// TIA Portal V20 export
DATA_BLOCK "Instance_FB_Digital_Output_DB"   // DB103
// stored: AutoNumber false, InstanceOfName FB_Digital_Output, InstanceOfType FB
"FB_Digital_Output"
   // VAR_INPUT
   //    DB_In_Emergency_Stop_Release : Bool;
   //    DB_In_Selected_Voltage_220V : Bool;
   //    DB_In_Selected_Voltage_127V : Bool;
   //    DB_Spin_Carousel_Frequency_Inverter_Speed_1 : Bool;
   //    DB_Spin_Carousel_Frequency_Inverter_Speed_2 : Bool;
   //    DB_Spin_Carousel_Frequency_Inverter_Speed_3 : Bool;
   //    DB_Conveyor_Belt_Frequency_Inverter_Speed_1 : Bool;
   //    DB_Conveyor_Belt_Frequency_Inverter_Speed_2 : Bool;
   //    DB_Conveyor_Belt_Frequency_Inverter_Speed_3 : Bool;
   //    DB_Turn_On_Conveyor_Belt_Motor_Spinner_Get_Entrace_Function_Test : Bool;
   //    DB_Turn_On_Conveyor_Belt_Motor_Rework_Conveyor_Belt_Get_Entrace_Functional_Test : Bool;
   //    DB_Turn_On_Conveyor_Belt_Motor_Spinner_Get_Exit_Functional_Test : Bool;
   //    DB_Turn_On_Conveyor_Belt_Motor_Rework_Conveyor_Belt_Get_Exit_Funcional_Test : Bool;
   //    DB_Open_Air_Pressure : Bool;
   //    DB_Valve_Advance_Spinner_Get_Entrace_Functional_Test : Bool;
   //    DB_Valve_Advance_Spinner_Get_Exit_Functional_Test : Bool;
   //    DB_Signal_Pre_Functional_Test_Production_Line : Bool;
   //    DB_Digital_Output_14 : Bool;
   //    DB_Digital_Output_15 : Bool;
   //    DB_Digital_Output_16 : Bool;
   //    DB_Digital_Output_17 : Bool;
   //    DB_Digital_Output_18 : Bool;
   //    DB_Digital_Output_19 : Bool;
   //    DB_Digital_Output_20 : Bool;
   //    DB_Digital_Output_21 : Bool;
   //    DB_Digital_Output_22 : Bool;
   //    DB_Digital_Output_23 : Bool;
   //    DB_Voltage_220V_Selected : Bool;
   //    DB_Voltage_127V_Selected : Bool;
   // END_VAR
   // VAR_OUTPUT
   //    DO_Spin_Carousel_Frequency_Inverter_Speed_1 : Bool;
   //    DO_Spin_Carousel_Frequency_Inverter_Speed_2 : Bool;
   //    DO_Spin_Carousel_Frequency_Inverter_Speed_3 : Bool;
   //    DO_Conveyor_Belt_Frequency_Inverter_Speed_1 : Bool;
   //    DO_Conveyor_Belt_Frequency_Inverter_Speed_2 : Bool;
   //    DO_Conveyor_Belt_Frequency_Inverter_Speed_3 : Bool;
   //    DO_Turn_On_Conveyor_Belt_Motor_Spinner_Get_Entrace_Function_Test : Bool;
   //    DO_Turn_On_Conveyor_Belt_Motor_Rework_Conveyor_Belt_Get_Entrace_Functional_Test : Bool;
   //    DO_Turn_On_Conveyor_Belt_Motor_Spinner_Get_Exit_Functional_Test : Bool;
   //    DO_Turn_On_Conveyor_Belt_Motor_Rework_Conveyor_Belt_Get_Exit_Funcional_Test : Bool;
   //    DO_Open_Air_Pressure : Bool;
   //    DO_Valve_Advance_Spinner_Entrace_Functional_Test : Bool;
   //    DO_Valve_Advance_Spinner_Exit_Functional_Test : Bool;
   //    DO_Signal_Pre_Functional_Test_Production_Line : Bool;
   //    DO_Digital_Output_14 : Bool;
   //    DO_Digital_Output_15 : Bool;
   //    DO_Digital_Output_16 : Bool;
   //    DO_Digital_Output_17 : Bool;
   //    DO_Digital_Output_18 : Bool;
   //    DO_Digital_Output_19 : Bool;
   //    DO_Digital_Output_20 : Bool;
   //    DO_Digital_Output_21 : Bool;
   //    DO_Digital_Output_22 : Bool;
   //    DO_Digital_Output_23 : Bool;
   //    DO_Voltage_220V_Selected : Bool;
   //    DO_Voltage_127V_Selected : Bool;
   // END_VAR
   // VAR
   //    Timer_Delay_Turn_On_220_V { S7_SetPoint := 'True'} : TON_TIME;
   //    Timer_Delay_Turn_On_127_V { S7_SetPoint := 'True'} : TON_TIME;
   // END_VAR
BEGIN
END_DATA_BLOCK
